// TIA Portal V20 export
// export: Created 2025-12-01T14:57:15.2889658Z, ExportSetting None, DisplayName Totally Integrated Automation Portal, DisplayVersion V20 Update 3, DisplayName TIA Portal Openness, DisplayVersion V20 Update 3, DisplayName TIA Portal Version Control Interface, DisplayVersion V20 Update 3, DisplayName STEP 7 Professional, DisplayVersion V20 Update 3, DisplayName STEP 7 Safety, DisplayVersion V20 Update 2, DisplayName WinCC Basic/Comfort/Advanced, DisplayVersion V20 Update 3, DisplayName WinCC Professional, DisplayVersion V20 Update 3, DisplayName WinCC Unified, DisplayVersion V20 Update 3
FUNCTION_BLOCK "FB910_CNT_UHS"   // FB910, LAD
{ S7_Optimized_Access := 'FALSE' }
// stored: AutoNumber false, SetENOAutomatically false
   VAR_INPUT
      IN { ExternalAccessible := 'False'; ExternalVisible := 'False'; ExternalWritable := 'False'} : Bool;   // Contar Tiempo
      R { ExternalAccessible := 'False'; ExternalVisible := 'False'; ExternalWritable := 'False'} : Bool;   // Resetear Tiempo
      PV { ExternalAccessible := 'False'; ExternalVisible := 'False'; ExternalWritable := 'False'} : Int;   // Valor a Contar (Unidades)
      BaseUnidades_ms : UDInt := 100;
   END_VAR
   VAR_OUTPUT
      QU : Bool;
      QD { ExternalAccessible := 'False'; ExternalVisible := 'False'; ExternalWritable := 'False'} : Bool;   // El tiempo se ha cumplido
      CVU : Int;   // Valor actual (Unidades)
      CVD : Int;   // Cuanto falta (Unidades)
   END_VAR
   VAR
      Valor_Actual { ExternalAccessible := 'False'; ExternalVisible := 'False'; ExternalWritable := 'False'} : DInt;
      STAT_Tiempo_OK { ExternalAccessible := 'False'; ExternalVisible := 'False'; ExternalWritable := 'False'} : Bool;
   END_VAR
   VAR_TEMP
      Aux_PV : DInt;
      Aux_CVU : DInt;
      Aux_CVD : DInt;
   END_VAR
BEGIN

REGION Network 1: Inicializar
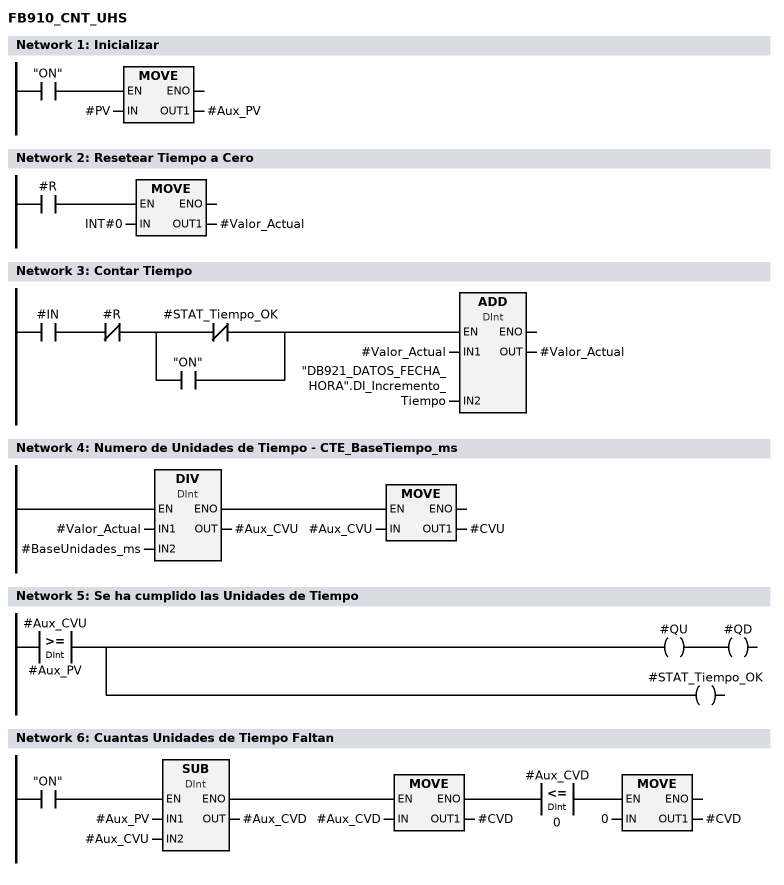
   RUNG wire#powerrail
      Contact( "ON" )
      Move(in := #PV, out1 => #Aux_PV)
   END_RUNG
   // the same network as SCL:
   IF "ON" THEN #Aux_PV := #PV; END_IF;
END_REGION

REGION Network 2: Resetear Tiempo a Cero
   RUNG wire#powerrail
      Contact( #R )
      { S7_GenerateENO := "TRUE" } Move(in := INT#0, out1 => #Valor_Actual)
   END_RUNG
   // the same network as SCL:
   IF #R THEN #Valor_Actual := INT#0; END_IF;
END_REGION

REGION Network 3: Contar Tiempo
   RUNG wire#powerrail
      Contact( #IN )
      I_Contact( #R )
      wire#w1
      I_Contact( #STAT_Tiempo_OK )
      wire#w2
      { S7_Templates := "SrcType := DInt"; S7_GenerateENO := "TRUE" } Add(in1 := #Valor_Actual, in2 := "DB921_DATOS_FECHA_HORA".DI_Incremento_Tiempo, out => #Valor_Actual)
   END_RUNG
   RUNG wire#w1
      Contact( "ON" )
   END_RUNG wire#w2
   // the same network as SCL:
   IF #IN AND NOT #R AND (NOT #STAT_Tiempo_OK OR "ON") THEN
       #Valor_Actual := #Valor_Actual + "DB921_DATOS_FECHA_HORA".DI_Incremento_Tiempo;
   END_IF;
END_REGION

REGION Network 4: Numero de Unidades de Tiempo - CTE_BaseTiempo_ms
   RUNG wire#powerrail
      { S7_Templates := "SrcType := DInt"; S7_GenerateENO := "TRUE" } Div(in1 := #Valor_Actual, in2 := #BaseUnidades_ms, out => #Aux_CVU)
      Move(in := #Aux_CVU, out1 => #CVU)
   END_RUNG
   // the same network as SCL:
   // ENO of a box is taken as its EN; it also drops when the box reports an error
   #Aux_CVU := #Valor_Actual / #BaseUnidades_ms;
   #CVU := #Aux_CVU;
END_REGION

REGION Network 5: Se ha cumplido las Unidades de Tiempo
   RUNG wire#powerrail
      { S7_Templates := "SrcType := DInt" } GE_Contact(in1 := #Aux_CVU, in2 := #Aux_PV)
      wire#w1
      Coil( #QU )
      Coil( #QD )
   END_RUNG
   RUNG wire#w1
      Coil( #STAT_Tiempo_OK )
   END_RUNG
   // the same network as SCL:
   #QU := #Aux_CVU >= #Aux_PV;
   #QD := #QU;
   #STAT_Tiempo_OK := #QU;
END_REGION

REGION Network 6: Cuantas Unidades de Tiempo Faltan
   RUNG wire#powerrail
      Contact( "ON" )
      { S7_Templates := "SrcType := DInt" } Sub(in1 := #Aux_PV, in2 := #Aux_CVU, out => #Aux_CVD)
      Move(in := #Aux_CVD, out1 => #CVD)
      { S7_Templates := "SrcType := DInt" } LE_Contact(in1 := #Aux_CVD, in2 := 0)
      Move(in := 0, out1 => #CVD)
   END_RUNG
   // the same network as SCL:
   IF "ON" THEN
       #Aux_CVD := #Aux_PV - #Aux_CVU;
       #CVD := #Aux_CVD;
   END_IF;
   IF "ON" AND (#Aux_CVD <= 0) THEN #CVD := 0; END_IF;
END_REGION
END_FUNCTION_BLOCK
